FUNCTION_BLOCK PickerSequence EXTENDS ZApplication.Sequence
VAR
  {attribute 'hide'}
  _parent : REFERENCE TO PickerUnit;
  _io : REFERENCE TO PickerIo;
  _actuator : REFERENCE TO PickerActuator;
  _fieldbus : REFERENCE TO PickerFieldbus;
  _axis : REFERENCE TO PickerAxis;
  _data : REFERENCE TO PickerDataRef;
  _unit : REFERENCE TO PickerLinkedUnit;  
END_VAR

METHOD FB_init : BOOL
VAR_INPUT
  bInitRetains : BOOL; // if TRUE, the retain variables are initialized (warm start / cold start)
  bInCopyCode : BOOL;  // if TRUE, the instance afterwards gets moved into the copy code (online change)
  unit : REFERENCE TO PickerUnit;
END_VAR
_parent REF= unit;
_alarming := unit._alarming;
_io REF= unit._equipment.Io;
_actuator REF= unit._equipment.Actuator;
_fieldbus REF= unit._equipment.Fieldbus;
_axis REF= unit._equipment.Axis;
_unit REF= unit._equipment.Unit;
_data REF= unit._data;
_loggerDiagnostics.SetLogger(unit._logger);
END_METHOD

METHOD StepDecoded : ZCore.ZString
VAR_INPUT
  stepIndex : INT;
END_VAR
VAR_INST
  _stepIndexDecoded : PickerStep;
END_VAR
_stepIndexDecoded := stepIndex;
stepDecoded := TO_STRING(_stepIndexDecoded);
END_METHOD

END_FUNCTION_BLOCK

(* stored: Version 1.1.0.1
   POU PickerSequence: Id {9c47d7b5-b342-48a2-b037-f6092a18a22b}, SpecialFunc None
   Method FB_init: Id {38ea3f80-55d5-46c9-b7ac-e6a5eed700d5}
   Method StepDecoded: Id {d33632e5-62f4-4052-b807-9ec2153234c9} *)
